{attribute addProperty BoxType "EP1122-0001-0018"}
{attribute addProperty Id "A_0027_EP1258_0001_0016EP1258_402FC40E44856A_0028_EP1258_0001_0017EP1258_402FC40E44856A_0029_EP1258_0001_0018EP1258_402FC40E44856A_0030_EP1258_0001_0019EP1258_402FC40E44856A_0031_EP1258_0001_0020EP1258_402FC40E44856A_0032_EP1258_0002_0016EP1258_402FC40E44856A_0033_EP1258_0002_0017EP1258_402FC40E44856A_0034_EP1258_0002_0018EP1258_402FC40E44856A_0035_EP1258_0002_0019EP1258_402FC40E44856A_0036_EP1258_0002_0020EP1258_402FC40E44856A_0037_EP1312_0001_0016A_0037_EP1312_0001_0016_F4B77AB8632068719477526"}
{attribute addProperty CRC "3507701713"}
{attribute addProperty SizeInBites "10800"}
{attribute addProperty SizeInBytes "68719478086"}
TYPE A_0026_EP1122_0001_0018_D11347D1 EXTENDS EP1122_179A0949 :
STRUCT
	{attribute addProperty Name "A_0027_EP1258_0001_0016"}
	A_0027_EP1258_0001_0016 : EP1258_402FC40E;
	{attribute addProperty Name "A_0028_EP1258_0001_0017"}
	A_0028_EP1258_0001_0017 : EP1258_402FC40E;
	{attribute addProperty Name "A_0029_EP1258_0001_0018"}
	A_0029_EP1258_0001_0018 : EP1258_402FC40E;
	{attribute addProperty Name "A_0030_EP1258_0001_0019"}
	A_0030_EP1258_0001_0019 : EP1258_402FC40E;
	{attribute addProperty Name "A_0031_EP1258_0001_0020"}
	A_0031_EP1258_0001_0020 : EP1258_402FC40E;
	{attribute addProperty Name "A_0032_EP1258_0002_0016"}
	A_0032_EP1258_0002_0016 : EP1258_402FC40E;
	{attribute addProperty Name "A_0033_EP1258_0002_0017"}
	A_0033_EP1258_0002_0017 : EP1258_402FC40E;
	{attribute addProperty Name "A_0034_EP1258_0002_0018"}
	A_0034_EP1258_0002_0018 : EP1258_402FC40E;
	{attribute addProperty Name "A_0035_EP1258_0002_0019"}
	A_0035_EP1258_0002_0019 : EP1258_402FC40E;
	{attribute addProperty Name "A_0036_EP1258_0002_0020"}
	A_0036_EP1258_0002_0020 : EP1258_402FC40E;
	{attribute addProperty Name "A_0037_EP1312_0001_0016"}
	A_0037_EP1312_0001_0016 : A_0037_EP1312_0001_0016_F4B77AB8;
END_STRUCT
END_TYPE

(* stored: Version 1.2.0.0, ProductVersion 3.1.4024.9
   DUT A_0026_EP1122_0001_0018_D11347D1: Id {951f4f8d-e7a1-49af-b195-feb6356e8c2d} *)
